// TIA Portal V21 export
TYPE "coneCrusherStopCtx"
   STRUCT
      "step" : USInt;
      stepTime : LTime;
      alm : "coneCrusherAlm";
      almDWord { S7_SetPoint := 'True'} : DWord;
   END_STRUCT;
END_TYPE
